TYPE ST_DiagHistory :
STRUCT
	nMaximum_Messages: BYTE;
	nNewest_Message: BYTE;
	nNewest_Acknowledged_Message: BYTE;
	bNewMessagesAvailable: BOOL;
	nFlags: UINT;
	DiagMessages: ARRAY[1..64] OF ST_DiagMessage;
END_STRUCT
END_TYPE

(* stored: Version 1.1.0.1, ProductVersion 3.1.4024.12
   DUT ST_DiagHistory: Id {e69c3287-5b6e-425b-87af-6759ae88f6cf} *)
